FUNCTION_BLOCK "SEQUENCE"   // FB18, GRAPH_PLUS
{ S7_Optimized_Access := 'TRUE' }
VERSION : 0.1
   VAR_INPUT
      OFF_SQ : Bool := false;   // Turn sequence off
      INIT_SQ : Bool := false;   // Set sequence to initial state
      ACK_EF : Bool := false;   // Acknowledge all errors and faults
      S_PREV : Bool := false;   // Output previous step in parameter S_NO
      S_NEXT : Bool := false;   // Indicate next step in parameter S_NO
      SW_AUTO : Bool := false;   // Automatic mode
      SW_TAP : Bool := false;   // Semiautomatic/switch with transition
      SW_TOP : Bool := false;   // Semiautomatic/ignore transition
      SW_MAN : Bool := false;   // Manual mode
      S_SEL : Int := 0;   // Select step to be output to S_NO
      S_ON : Bool := false;   // Activate step indicated in S_NO
      S_OFF : Bool := false;   // Deactivate step indicated S_NO
      T_PUSH : Bool := false;   // Enable transition to switch in semi automatic mode
   END_VAR
   VAR_OUTPUT
      S_NO : Int := 0;   // Step number
      S_MORE : Bool := false;   // More steps are available and can be shown in S_NO
      S_ACTIVE : Bool := false;   // Step indicated in S_NO is active
      ERR_FLT : Bool := false;   // Interlock or supervision group error
      AUTO_ON : Bool := false;   // Automatic mode is active
      TAP_ON : Bool := false;   // Semiautomatic mode/step with transition enabled
      TOP_ON : Bool := false;   // Semiautomatic mode/ignore transition enabled
      MAN_ON : Bool := false;   // Manual mode is active
   END_VAR
   VAR
      HMI_INFO : Array[0..8] of UInt;
      IF_PAR : G7_IfParPlus_V2;
      RT_DATA : G7_RTDataPlus_V2;   // Internal data area
      Trans1 : G7_TransitionPlus_V2;   // Transition structure
      Trans2 : G7_TransitionPlus_V2;   // Transition structure
      Trans3 : G7_TransitionPlus_V2;   // Transition structure
      Trans4 : G7_TransitionPlus_V2;   // Transition structure
      Trans5 : G7_TransitionPlus_V2;   // Transition structure
      Idle : G7_StepPlus_V2;   // Step structure
      Warmup : G7_StepPlus_V2;   // Step structure
      Stabilize : G7_StepPlus_V2;   // Step structure
      Generation : G7_StepPlus_V2;   // Step structure
      Cooldown : G7_StepPlus_V2;   // Step structure
      SINI : Array[0..1] of USInt;
      LSTT : Array[0..4] of USInt;
      ATAJ : Array[0..4] of USInt;
      ATAB : Array[0..4] of USInt;
      PSTT : Array[0..4] of USInt;
      NSTT : Array[0..4] of USInt;
      ASSJ : Array[0..4] of USInt;
      ASSB : Array[0..4] of USInt;
      PTTS : Array[0..4] of USInt;
      NTTS : Array[0..4] of USInt;
      SW_SQTS : Array[0..4] of USInt;
      SWITCH : Array[0..0] of USInt;
      TVX : Array[0..1] of USInt;
      TTX : Array[0..1] of USInt;
      TSX : Array[0..1] of USInt;
      S00X : Array[0..1] of USInt;
      SOFFX : Array[0..1] of USInt;
      SONX : Array[0..1] of USInt;
      SAX : Array[0..1] of USInt;
      SERRX : Array[0..5] of USInt;
      SMX : Array[0..5] of USInt;
      S0X : Array[0..5] of USInt;
      S1X : Array[0..5] of USInt;
      IL_ALARM_INST : Program_Alarm;
      SUP_ALARM_INST : Program_Alarm;
      STEP_TIME_ALARM_INST : Program_Alarm;
      IEC_TIMER_INST : IEC_TIMER;
      TRANSACTION_FLAG : Bool := false;
   END_VAR
   // SINI[0] := 2;
   // LSTT[0] := 255;
   // LSTT[1] := 255;
   // LSTT[2] := 255;
   // LSTT[3] := 255;
   // ATAJ[1] := 1;
   // ATAJ[2] := 2;
   // ATAJ[3] := 3;
   // ATAJ[4] := 4;
   // ATAB[1] := 1;
   // ATAB[2] := 2;
   // ATAB[3] := 3;
   // ATAB[4] := 4;
   // PSTT[1] := 1;
   // PSTT[2] := 2;
   // PSTT[3] := 3;
   // PSTT[4] := 4;
   // NSTT[0] := 1;
   // NSTT[1] := 2;
   // NSTT[2] := 3;
   // NSTT[3] := 4;
   // ASSJ[1] := 1;
   // ASSJ[2] := 2;
   // ASSJ[3] := 3;
   // ASSJ[4] := 4;
   // ASSB[1] := 1;
   // ASSB[2] := 2;
   // ASSB[3] := 3;
   // ASSB[4] := 4;
   // PTTS[0] := 255;
   // PTTS[2] := 1;
   // PTTS[3] := 2;
   // PTTS[4] := 3;
   // NTTS[1] := 1;
   // NTTS[2] := 2;
   // NTTS[3] := 3;
   // NTTS[4] := 4;
   // TVX[0] := 16#1;
   // TTX[0] := 16#1;
   // TSX[0] := 16#1;
   // S00X[0] := 16#1;
   // SOFFX[0] := 16#1;
   // SONX[0] := 16#1;
   // SAX[0] := 16#1;
   // SERRX[0] := 16#1;
   // SMX[0] := 16#1;
   // S0X[0] := 16#1;
   // S1X[0] := 16#1;
BEGIN
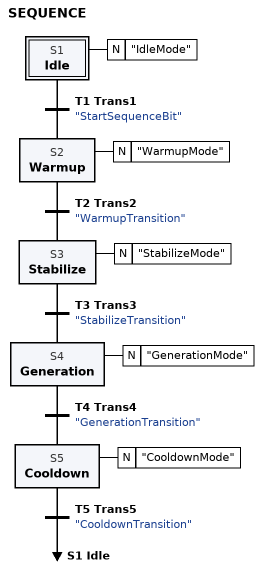
   // sequencer 1
   INITIAL_STEP Idle:   // S1, max time T#10S, warning time T#7S
              N    "IdleMode"
   END_STEP
   TRANSITION Trans1 FROM Idle TO Warmup   // T1
      := "StartSequenceBit";
   END_TRANSITION
   STEP Warmup:   // S2, max time T#10S, warning time T#7S
              N    "WarmupMode"
   END_STEP
   TRANSITION Trans2 FROM Warmup TO Stabilize   // T2
      := "WarmupTransition";
   END_TRANSITION
   STEP Stabilize:   // S3, max time T#10S, warning time T#7S
              N    "StabilizeMode"
   END_STEP
   TRANSITION Trans3 FROM Stabilize TO Generation   // T3
      := "StabilizeTransition";
   END_TRANSITION
   STEP Generation:   // S4, max time T#10S, warning time T#7S
              N    "GenerationMode"
   END_STEP
   TRANSITION Trans4 FROM Generation TO Cooldown   // T4
      := "GenerationTransition";
   END_TRANSITION
   STEP Cooldown:   // S5, max time T#10S, warning time T#7S
              N    "CooldownMode"
   END_STEP
   TRANSITION Trans5 FROM Cooldown TO Idle   // T5, jump
      := "CooldownTransition";
   END_TRANSITION
END_FUNCTION_BLOCK

FUNCTION_BLOCK "HOURMETER_LAD"   // FB19, LAD
{ S7_Optimized_Access := 'TRUE' }
VERSION : 0.1
   VAR
      Accum_Elapsed : Time;
      OS1 : Bool;
      MinuteTimedDown : Bool;
      HourCountedDown : Bool;
      OS2 : Bool;
      OS3 : Bool;
      DayCountedDown : Bool;
      ResetTime : Time;
      OS4 : Bool;
      ResetRTO : Bool;
      MinuteCounterReset : Bool;
      HourCounterReset : Bool;
   END_VAR
   VAR_TEMP
      ResetHourmeterTrigger : Bool;
   END_VAR
   VAR_TEMP   // added for the SCL form of the ladder/FBD networks
      _w1 : Bool;
      _w2 : Bool;
      _w3 : Bool;
   END_VAR
BEGIN

REGION Network 1
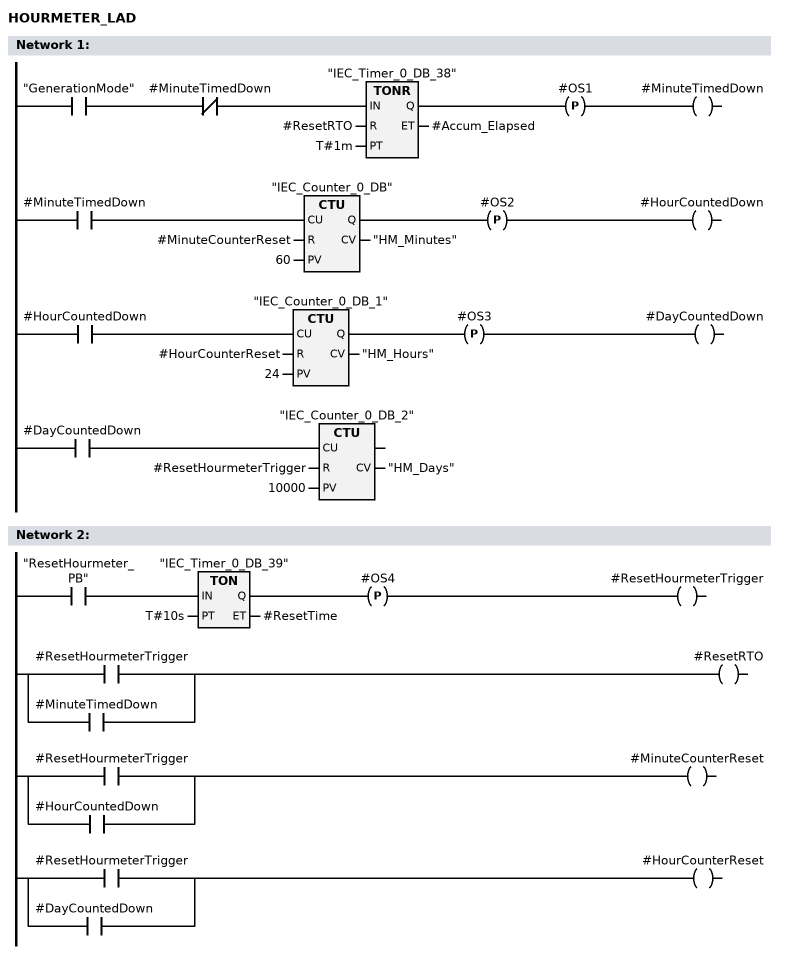
   "IEC_Timer_0_DB_38".TONR(IN := "GenerationMode" AND NOT #MinuteTimedDown,
                           R := #ResetRTO,
                           PT := T#1m,
                           ET => #Accum_Elapsed);
   #_w1 := "IEC_Timer_0_DB_38".Q AND NOT #OS1;   // rising edge
   #OS1 := "IEC_Timer_0_DB_38".Q;
   #MinuteTimedDown := #_w1;
   "IEC_Counter_0_DB".CTU(CU := #MinuteTimedDown, R := #MinuteCounterReset, PV := 60, CV => "HM_Minutes");
   #_w2 := "IEC_Counter_0_DB".Q AND NOT #OS2;   // rising edge
   #OS2 := "IEC_Counter_0_DB".Q;
   #HourCountedDown := #_w2;
   "IEC_Counter_0_DB_1".CTU(CU := #HourCountedDown, R := #HourCounterReset, PV := 24, CV => "HM_Hours");
   #_w3 := "IEC_Counter_0_DB_1".Q AND NOT #OS3;   // rising edge
   #OS3 := "IEC_Counter_0_DB_1".Q;
   #DayCountedDown := #_w3;
   "IEC_Counter_0_DB_2".CTU(CU := #DayCountedDown, R := #ResetHourmeterTrigger, PV := 10000, CV => "HM_Days");
END_REGION

REGION Network 2
   "IEC_Timer_0_DB_39".TON(IN := "ResetHourmeter_PB", PT := T#10s, ET => #ResetTime);
   #_w1 := "IEC_Timer_0_DB_39".Q AND NOT #OS4;   // rising edge
   #OS4 := "IEC_Timer_0_DB_39".Q;
   #ResetHourmeterTrigger := #_w1;
   #ResetRTO := #ResetHourmeterTrigger OR #MinuteTimedDown;
   #MinuteCounterReset := #ResetHourmeterTrigger OR #HourCountedDown;
   #HourCounterReset := #ResetHourmeterTrigger OR #DayCountedDown;
END_REGION
END_FUNCTION_BLOCK

FUNCTION_BLOCK "HOURMETER_FBD"   // FB20, FBD
{ S7_Optimized_Access := 'TRUE' }
VERSION : 0.1
   VAR
      Accum_Elapsed : Time;
      OS1 : Bool;
      MinuteTimedDown : Bool;
      HourCountedDown : Bool;
      OS2 : Bool;
      OS3 : Bool;
      DayCountedDown : Bool;
      ResetTime : Time;
      OS4 : Bool;
      ResetRTO : Bool;
      MinuteCounterReset : Bool;
      HourCounterReset : Bool;
   END_VAR
   VAR_TEMP
      ResetHourmeterTrigger : Bool;
   END_VAR
   VAR_TEMP   // added for the SCL form of the ladder/FBD networks
      _w1 : Bool;
      _w2 : Bool;
      _w3 : Bool;
   END_VAR
BEGIN

REGION Network 1
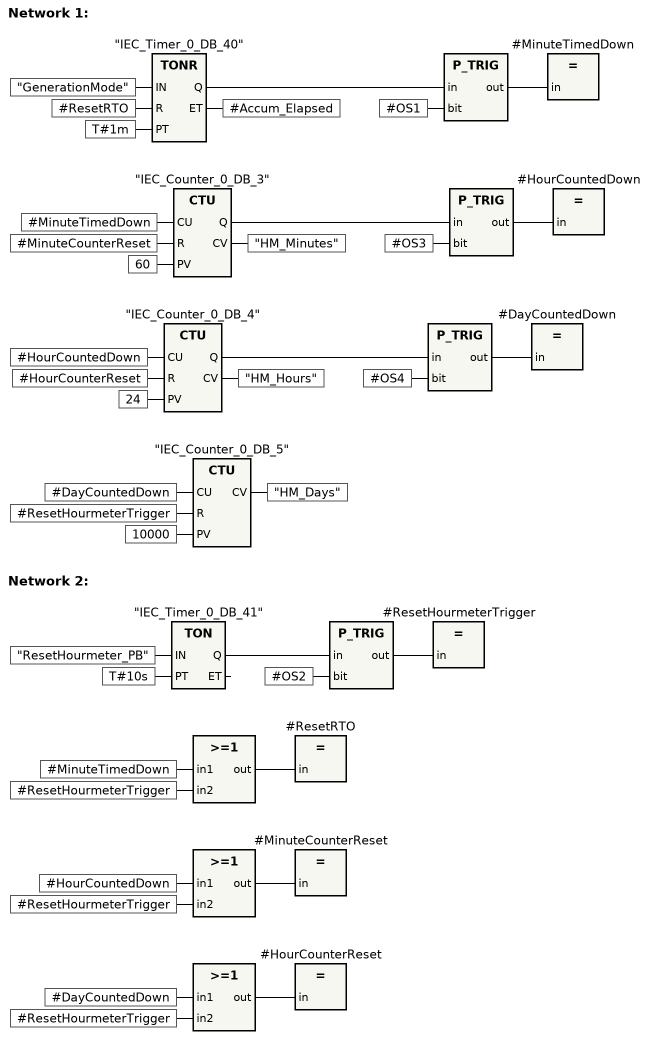
   "IEC_Timer_0_DB_40".TONR(IN := "GenerationMode", R := #ResetRTO, PT := T#1m, ET => #Accum_Elapsed);
   #_w1 := "IEC_Timer_0_DB_40".Q AND NOT #OS1;   // rising edge
   #OS1 := "IEC_Timer_0_DB_40".Q;
   #MinuteTimedDown := #_w1;
   "IEC_Counter_0_DB_3".CTU(CU := #MinuteTimedDown, R := #MinuteCounterReset, PV := 60, CV => "HM_Minutes");
   #_w2 := "IEC_Counter_0_DB_3".Q AND NOT #OS3;   // rising edge
   #OS3 := "IEC_Counter_0_DB_3".Q;
   #HourCountedDown := #_w2;
   "IEC_Counter_0_DB_4".CTU(CU := #HourCountedDown, R := #HourCounterReset, PV := 24, CV => "HM_Hours");
   #_w3 := "IEC_Counter_0_DB_4".Q AND NOT #OS4;   // rising edge
   #OS4 := "IEC_Counter_0_DB_4".Q;
   #DayCountedDown := #_w3;
   "IEC_Counter_0_DB_5".CTU(CU := #DayCountedDown, R := #ResetHourmeterTrigger, PV := 10000, CV => "HM_Days");
END_REGION

REGION Network 2
   "IEC_Timer_0_DB_41".TON(IN := "ResetHourmeter_PB", PT := T#10s);
   #_w1 := "IEC_Timer_0_DB_41".Q AND NOT #OS2;   // rising edge
   #OS2 := "IEC_Timer_0_DB_41".Q;
   #ResetHourmeterTrigger := #_w1;
   #ResetRTO := #MinuteTimedDown OR #ResetHourmeterTrigger;
   #MinuteCounterReset := #HourCountedDown OR #ResetHourmeterTrigger;
   #HourCounterReset := #DayCountedDown OR #ResetHourmeterTrigger;
END_REGION
END_FUNCTION_BLOCK

FUNCTION_BLOCK "HOURMETER_SCL"   // FB21, SCL
{ S7_Optimized_Access := 'TRUE' }
VERSION : 0.1
   VAR
      Accum_Elapsed : Time;
      OS1 : Bool;
      MinuteTimedDown : Bool;
      HourCountedDown : Bool;
      OS2 : Bool;
      OS3 : Bool;
      DayCountedDown : Bool;
      ResetTime : Time;
      OS4 : Bool;
      ResetRTO : Bool;
      MinuteCounterReset : Bool;
      HourCounterReset : Bool;
   END_VAR
   VAR_TEMP
      ResetHourmeterTrigger : Bool;
   END_VAR
BEGIN
   IF "GenerationMode" THEN
       "IEC_Timer_0_DB_43".TONR(IN := TRUE,
                                R := #ResetRTO,
                                PT := T#60s,
                                Q => #MinuteTimedDown,
                                ET => #Accum_Elapsed);
   END_IF;

   IF #MinuteTimedDown THEN
       RESET_TIMER("IEC_Timer_0_DB_43");
   END_IF;

   "IEC_Counter_0_DB_6".CTU(CU:=#MinuteTimedDown,
                            R:=#MinuteCounterReset,
                            PV:=60,
                            Q=>#HourCountedDown,
                            CV=>"HM_Minutes");

   "IEC_Counter_0_DB_7".CTU(CU:=#HourCountedDown,
                            R:=#HourCounterReset,
                            PV:=24,
                            Q=>#DayCountedDown,
                            CV=>"HM_Hours");

   "IEC_Counter_0_DB_8".CTU(CU:=#DayCountedDown,
                            R:=#ResetHourmeterTrigger,
                            PV:=10000,
                            CV=>"HM_Days");

   IF "ResetHourmeter_PB" THEN
       "IEC_Timer_0_DB_44".TON(IN := TRUE,
                               PT := T#10s,
                               Q => #ResetHourmeterTrigger);
   ELSE
       RESET_TIMER("IEC_Timer_0_DB_44");
   END_IF;

   IF #ResetHourmeterTrigger OR #MinuteTimedDown THEN
       #ResetRTO := 1;
   ELSE
       #ResetRTO := 0;
   END_IF;

   IF #ResetHourmeterTrigger OR #HourCountedDown THEN
       #MinuteCounterReset := 1;
   ELSE
       #MinuteCounterReset := 0;
   END_IF;

   IF #ResetHourmeterTrigger OR #DayCountedDown THEN
       #HourCounterReset := 1;
   ELSE
       #HourCounterReset := 0;
   END_IF;
END_FUNCTION_BLOCK

FUNCTION_BLOCK "HOURMETER_STL"   // FB22, STL
{ S7_Optimized_Access := 'TRUE' }
VERSION : 0.1
   VAR
      Accum_Elapsed : Time;
      OS1 : Bool;
      MinuteTimedDown : Bool;
      HourCountedDown : Bool;
      OS2 : Bool;
      OS3 : Bool;
      DayCountedDown : Bool;
      ResetTime : Time;
      OS4 : Bool;
      ResetRTO : Bool;
      MinuteCounterReset : Bool;
      HourCounterReset : Bool;
   END_VAR
   VAR_TEMP
      ResetHourmeterTrigger : Bool;
      TooManyDays : Bool;
      Acc_Time : Time;
   END_VAR
BEGIN

REGION Network 1
         A     "GenerationMode";
         JC    RTOTimer;
         CLR;
         JU    EndOfLine;

   RTOTimer:CALL  TONR, "IEC_Timer_0_DB_45"
         ( IN := TRUE,
           R  := #ResetRTO,
           PT := T#1m,
           Q  := #MinuteTimedDown,
           ET := #Accum_Elapsed
         );

         CALL  CTU, "IEC_Counter_0_DB_9"
         ( CU := #MinuteTimedDown,
           R  := #MinuteCounterReset,
           PV := 60,
           Q  := #HourCountedDown,
           CV := "HM_Minutes"
         );

         CALL  CTU, "IEC_Counter_0_DB_10"
         ( CU := #HourCountedDown,
           R  := #HourCounterReset,
           PV := 24,
           Q  := #DayCountedDown,
           CV := "HM_Hours"
         );

         CALL  CTU, "IEC_Counter_0_DB_11"
         ( CU := #DayCountedDown,
           R  := #ResetHourmeterTrigger,
           PV := 10000,
           Q  := #TooManyDays,
           CV := "HM_Days"
         );

         JU    EndOfLine;



   ResetEvaluate:CLR;
         A     "ResetHourmeter_PB";
         JC    ResetHourmeter;
         CALL  RESET_TIMER
         ( "TIMER" := "IEC_Timer_0_DB_46"
         );
         JU    EndOfLine;

   ResetHourmeter:CALL  TON, "IEC_Timer_0_DB_46"
         ( IN := TRUE,
           PT := T#10s,
           Q  := #ResetHourmeterTrigger,
           ET := #Acc_Time
         );

   EndOfLine:A     #ResetHourmeterTrigger;
         O     #MinuteTimedDown;
         =     #ResetRTO;
         CLR;
         A     #ResetHourmeterTrigger;
         O     #HourCountedDown;
         =     #MinuteCounterReset;
         CLR;
         A     #ResetHourmeterTrigger;
         O     #DayCountedDown;
         =     #HourCountedDown;
END_REGION
END_FUNCTION_BLOCK

FUNCTION "SCP" : Void   // FC1, FBD
{ S7_Optimized_Access := 'TRUE' }
VERSION : 0.1
   VAR_INPUT
      Input_Min : Int;
      Input_Max : Int;
      Input_Signal : Int;
      Output_Min : Int;
      Output_Max : Int;
   END_VAR
   VAR_OUTPUT
      SV : Int;
   END_VAR
   VAR_TEMP
      TV : Real;
   END_VAR
BEGIN

REGION Network 1
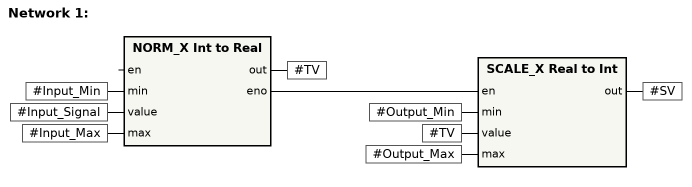
   #TV := NORM_X(MIN := #Input_Min, VALUE := #Input_Signal, MAX := #Input_Max);
   #SV := SCALE_X(MIN := #Output_Min, VALUE := #TV, MAX := #Output_Max);
END_REGION
END_FUNCTION

FUNCTION "MOVE" : Void   // FC2, FBD
{ S7_Optimized_Access := 'TRUE' }
VERSION : 0.1
   VAR_INPUT
      Int1 : Int;
   END_VAR
   VAR_OUTPUT
      Time1 : Time;
   END_VAR
   VAR_TEMP
      TV : Int;
   END_VAR
BEGIN

REGION Network 1
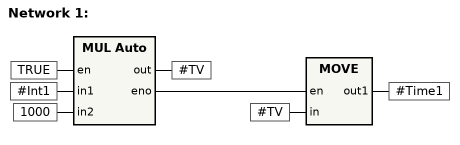
   IF TRUE THEN
       #TV := #Int1 * 1000;
       #Time1 := #TV;
   END_IF;
END_REGION
END_FUNCTION

ORGANIZATION_BLOCK "Main"   // OB1, LAD, ProgramCycle
TITLE = "Main Program Sweep (Cycle)"
{ S7_Optimized_Access := 'TRUE' }
VERSION : 0.1
   VAR_INPUT
      Initial_Call : Bool;   // Initial call of this OB
      Remanence : Bool;   // =True, if remanent data are available
   END_VAR
   VAR_TEMP
      SequenceInit : Bool;
      InitSequence : Bool;
   END_VAR
   VAR_TEMP   // added for the SCL form of the ladder/FBD networks
      _w1 : Bool;
      _w2 : Bool;
      _w3 : Bool;
      _w4 : Bool;
   END_VAR
BEGIN

REGION Network 1
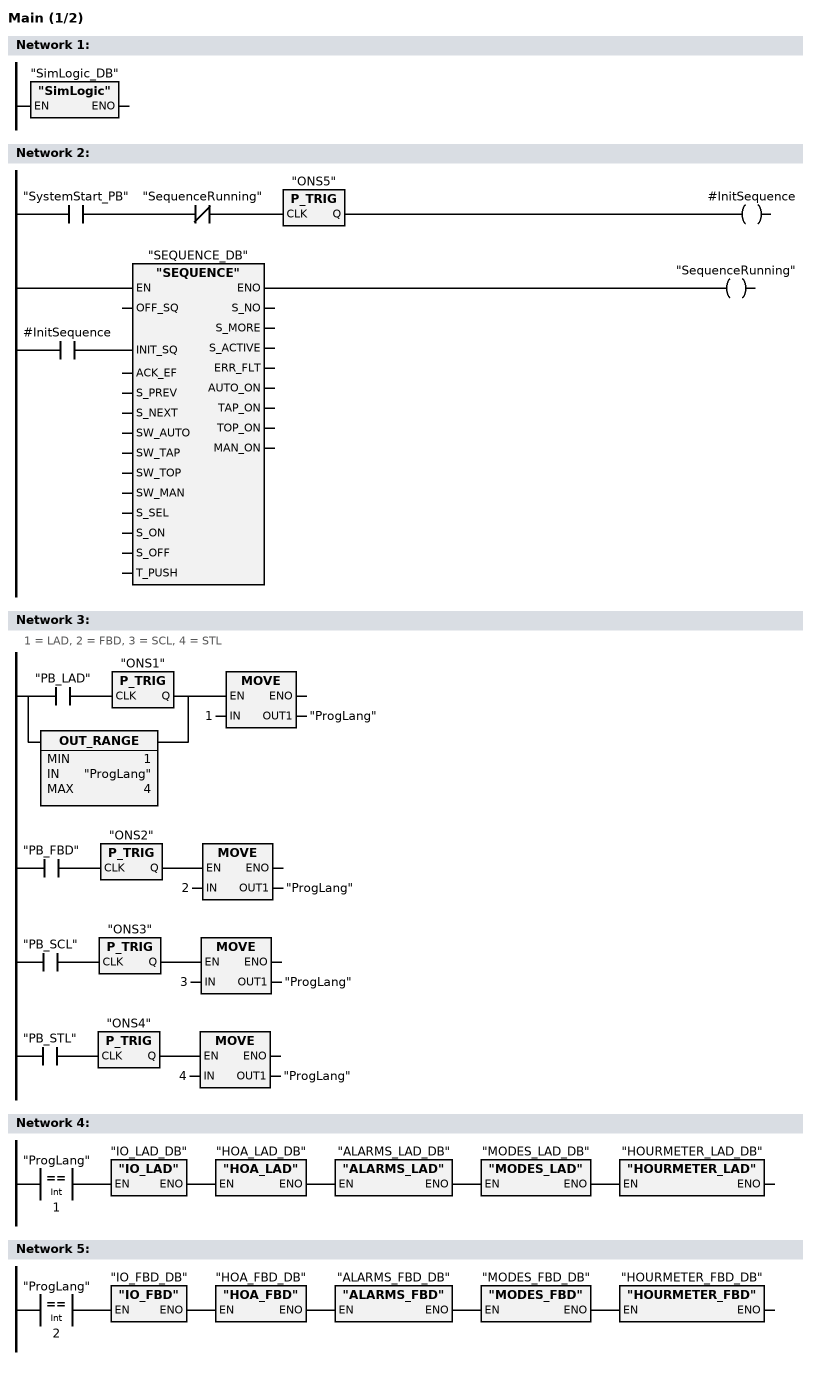
   RUNG wire#powerrail
      "SimLogic_DB"()
   END_RUNG
   // the same network as SCL:
   "SimLogic_DB"();   // "SimLogic"
END_REGION

REGION Network 2
   RUNG wire#powerrail
      Contact( "SystemStart_PB" )
      I_Contact( "SequenceRunning" )
      P_Trig( "ONS5" )
      Coil( #InitSequence )
   END_RUNG
   RUNG wire#powerrail
      "SEQUENCE_DB"(INIT_SQ := wire#w1, OFF_SQ :=, ACK_EF :=, S_PREV :=, S_NEXT :=, SW_AUTO :=, SW_TAP :=, SW_TOP :=, SW_MAN :=, S_SEL :=, S_ON :=, S_OFF :=, T_PUSH :=, S_NO =>, S_MORE =>, S_ACTIVE =>, ERR_FLT =>, AUTO_ON =>, TAP_ON =>, TOP_ON =>, MAN_ON =>)
      Coil( "SequenceRunning" )
   END_RUNG
   RUNG wire#powerrail
      Contact( #InitSequence )
   END_RUNG wire#w1
   // the same network as SCL:
   #_w1 := "SystemStart_PB" AND NOT "SequenceRunning";
   #_w2 := #_w1 AND NOT "ONS5";   // rising edge
   "ONS5" := #_w1;
   #InitSequence := #_w2;
   "SEQUENCE_DB"(INIT_SQ := #InitSequence, ENO => #_w3);   // "SEQUENCE"
   "SequenceRunning" := #_w3;
END_REGION

REGION Network 3
   // 1 = LAD, 2 = FBD, 3 = SCL, 4 = STL
   #_w1 := "PB_LAD" AND NOT "ONS1";   // rising edge
   "ONS1" := "PB_LAD";
   IF #_w1 OR ("ProgLang" < 1) OR ("ProgLang" > 4) THEN "ProgLang" := 1; END_IF;
   #_w2 := "PB_FBD" AND NOT "ONS2";   // rising edge
   "ONS2" := "PB_FBD";
   IF #_w2 THEN "ProgLang" := 2; END_IF;
   #_w3 := "PB_SCL" AND NOT "ONS3";   // rising edge
   "ONS3" := "PB_SCL";
   IF #_w3 THEN "ProgLang" := 3; END_IF;
   #_w4 := "PB_STL" AND NOT "ONS4";   // rising edge
   "ONS4" := "PB_STL";
   IF #_w4 THEN "ProgLang" := 4; END_IF;
END_REGION

REGION Network 4
   RUNG wire#powerrail
      { S7_Templates := "SrcType := Int" } EQ_Contact(in1 := "ProgLang", in2 := 1)
      "IO_LAD_DB"()
      "HOA_LAD_DB"()
      "ALARMS_LAD_DB"()
      "MODES_LAD_DB"()
      "HOURMETER_LAD_DB"()
   END_RUNG
   // the same network as SCL:
   "IO_LAD_DB"(EN := "ProgLang" = 1, ENO => #_w1);   // "IO_LAD"
   "HOA_LAD_DB"(EN := #_w1, ENO => #_w2);   // "HOA_LAD"
   "ALARMS_LAD_DB"(EN := #_w2, ENO => #_w3);   // "ALARMS_LAD"
   "MODES_LAD_DB"(EN := #_w3, ENO => #_w4);   // "MODES_LAD"
   IF #_w4 THEN
       "HOURMETER_LAD_DB"();   // "HOURMETER_LAD"
   END_IF;
END_REGION

REGION Network 5
   RUNG wire#powerrail
      { S7_Templates := "SrcType := Int" } EQ_Contact(in1 := "ProgLang", in2 := 2)
      "IO_FBD_DB"()
      "HOA_FBD_DB"()
      "ALARMS_FBD_DB"()
      "MODES_FBD_DB"()
      "HOURMETER_FBD_DB"()
   END_RUNG
   // the same network as SCL:
   "IO_FBD_DB"(EN := "ProgLang" = 2, ENO => #_w1);   // "IO_FBD"
   "HOA_FBD_DB"(EN := #_w1, ENO => #_w2);   // "HOA_FBD"
   "ALARMS_FBD_DB"(EN := #_w2, ENO => #_w3);   // "ALARMS_FBD"
   "MODES_FBD_DB"(EN := #_w3, ENO => #_w4);   // "MODES_FBD"
   IF #_w4 THEN
       "HOURMETER_FBD_DB"();   // "HOURMETER_FBD"
   END_IF;
END_REGION

REGION Network 6
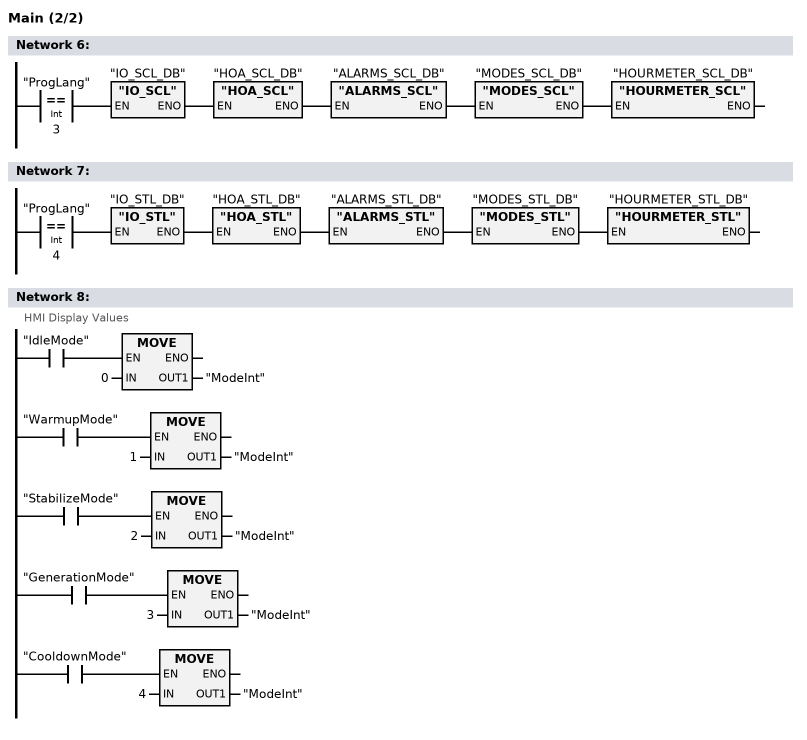
   RUNG wire#powerrail
      { S7_Templates := "SrcType := Int" } EQ_Contact(in1 := "ProgLang", in2 := 3)
      "IO_SCL_DB"()
      "HOA_SCL_DB"()
      "ALARMS_SCL_DB"()
      "MODES_SCL_DB"()
      "HOURMETER_SCL_DB"()
   END_RUNG
   // the same network as SCL:
   "IO_SCL_DB"(EN := "ProgLang" = 3, ENO => #_w1);   // "IO_SCL"
   "HOA_SCL_DB"(EN := #_w1, ENO => #_w2);   // "HOA_SCL"
   "ALARMS_SCL_DB"(EN := #_w2, ENO => #_w3);   // "ALARMS_SCL"
   "MODES_SCL_DB"(EN := #_w3, ENO => #_w4);   // "MODES_SCL"
   IF #_w4 THEN
       "HOURMETER_SCL_DB"();   // "HOURMETER_SCL"
   END_IF;
END_REGION

REGION Network 7
   RUNG wire#powerrail
      { S7_Templates := "SrcType := Int" } EQ_Contact(in1 := "ProgLang", in2 := 4)
      "IO_STL_DB"()
      "HOA_STL_DB"()
      "ALARMS_STL_DB"()
      "MODES_STL_DB"()
      "HOURMETER_STL_DB"()
   END_RUNG
   // the same network as SCL:
   "IO_STL_DB"(EN := "ProgLang" = 4, ENO => #_w1);   // "IO_STL"
   "HOA_STL_DB"(EN := #_w1, ENO => #_w2);   // "HOA_STL"
   "ALARMS_STL_DB"(EN := #_w2, ENO => #_w3);   // "ALARMS_STL"
   "MODES_STL_DB"(EN := #_w3, ENO => #_w4);   // "MODES_STL"
   IF #_w4 THEN
       "HOURMETER_STL_DB"();   // "HOURMETER_STL"
   END_IF;
END_REGION

REGION Network 8
   // HMI Display Values
   RUNG wire#powerrail
      Contact( "IdleMode" )
      Move(in := 0, out1 => "ModeInt")
   END_RUNG
   RUNG wire#powerrail
      Contact( "WarmupMode" )
      Move(in := 1, out1 => "ModeInt")
   END_RUNG
   RUNG wire#powerrail
      Contact( "StabilizeMode" )
      Move(in := 2, out1 => "ModeInt")
   END_RUNG
   RUNG wire#powerrail
      Contact( "GenerationMode" )
      Move(in := 3, out1 => "ModeInt")
   END_RUNG
   RUNG wire#powerrail
      Contact( "CooldownMode" )
      Move(in := 4, out1 => "ModeInt")
   END_RUNG
   // the same network as SCL:
   IF "IdleMode" THEN "ModeInt" := 0; END_IF;
   IF "WarmupMode" THEN "ModeInt" := 1; END_IF;
   IF "StabilizeMode" THEN "ModeInt" := 2; END_IF;
   IF "GenerationMode" THEN "ModeInt" := 3; END_IF;
   IF "CooldownMode" THEN "ModeInt" := 4; END_IF;
END_REGION
END_ORGANIZATION_BLOCK

ORGANIZATION_BLOCK "PID"   // OB30, LAD, CyclicInterrupt
{ S7_Optimized_Access := 'TRUE' }
VERSION : 0.1
   VAR_INPUT
      Initial_Call : Bool;   // Initial call of this OB
      Event_Count : Int;   // Events discarded
   END_VAR
   VAR_TEMP
      BSP : Real;
      VSP : Real;
      BaffleHandTrigger : Bool;
      BaffleAutoTrigger : Bool;
      BaffleOffTrigger : Bool;
      VFDHandTrigger : Bool;
      VFDOffTrigger : Bool;
      VFDAutoTrigger : Bool;
   END_VAR
   VAR_TEMP   // added for the SCL form of the ladder/FBD networks
      _w1 : Bool;
      _w2 : Bool;
      _w3 : Bool;
      _w4 : Bool;
      _w5 : Bool;
      _w6 : Bool;
      _w7 : Bool;
   END_VAR
BEGIN

REGION Network 1: Oil High Flow Alarm Handling
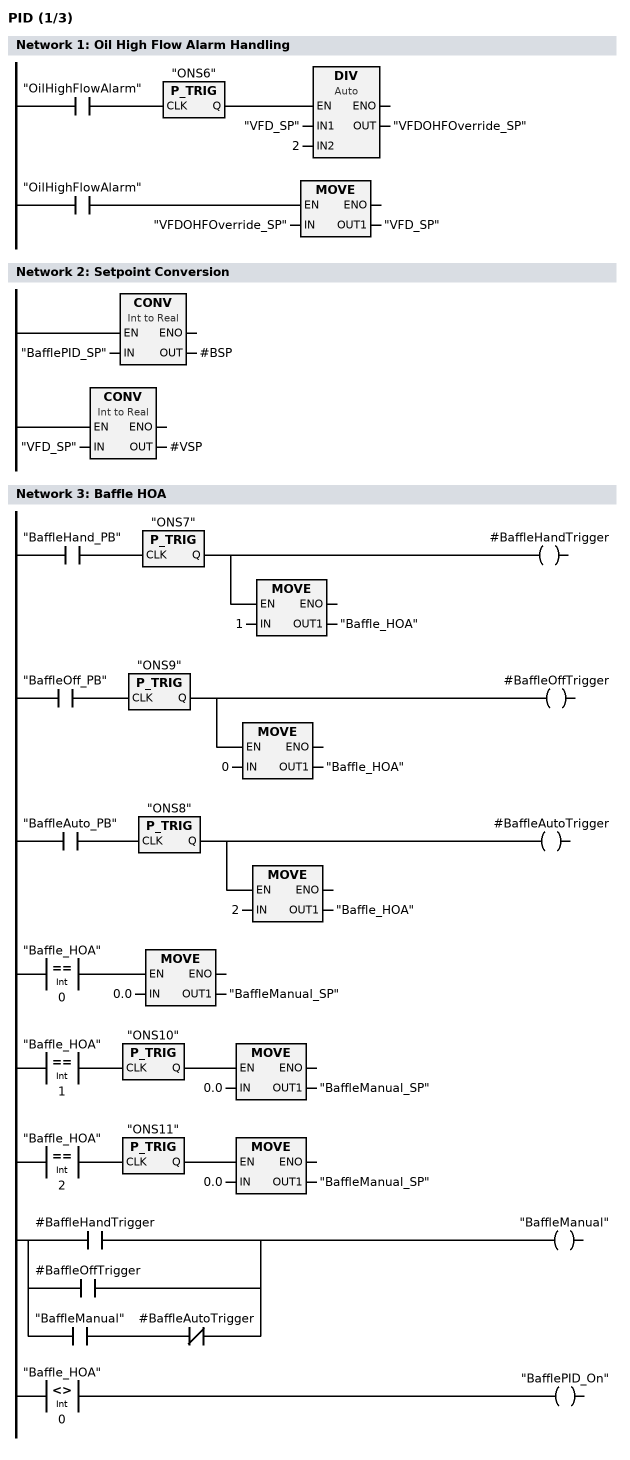
   RUNG wire#powerrail
      Contact( "OilHighFlowAlarm" )
      P_Trig( "ONS6" )
      Div(in1 := "VFD_SP", in2 := 2, out => "VFDOHFOverride_SP")
   END_RUNG
   RUNG wire#powerrail
      Contact( "OilHighFlowAlarm" )
      Move(in := "VFDOHFOverride_SP", out1 => "VFD_SP")
   END_RUNG
   // the same network as SCL:
   #_w1 := "OilHighFlowAlarm" AND NOT "ONS6";   // rising edge
   "ONS6" := "OilHighFlowAlarm";
   IF #_w1 THEN "VFDOHFOverride_SP" := "VFD_SP" / 2; END_IF;
   IF "OilHighFlowAlarm" THEN "VFD_SP" := "VFDOHFOverride_SP"; END_IF;
END_REGION

REGION Network 2: Setpoint Conversion
   RUNG wire#powerrail
      { S7_Templates := "[SrcType := Int, DestType := Real]" } Convert(in := "BafflePID_SP", out => #BSP)
   END_RUNG
   RUNG wire#powerrail
      { S7_Templates := "[SrcType := Int, DestType := Real]" } Convert(in := "VFD_SP", out => #VSP)
   END_RUNG
   // the same network as SCL:
   #BSP := INT_TO_REAL("BafflePID_SP");
   #VSP := INT_TO_REAL("VFD_SP");
END_REGION

REGION Network 3: Baffle HOA
   RUNG wire#powerrail
      Contact( "BaffleHand_PB" )
      P_Trig( "ONS7" )
      wire#w1
      Coil( #BaffleHandTrigger )
   END_RUNG
   RUNG wire#w1
      Move(in := 1, out1 => "Baffle_HOA")
   END_RUNG
   RUNG wire#powerrail
      Contact( "BaffleOff_PB" )
      P_Trig( "ONS9" )
      wire#w2
      Coil( #BaffleOffTrigger )
   END_RUNG
   RUNG wire#w2
      Move(in := 0, out1 => "Baffle_HOA")
   END_RUNG
   RUNG wire#powerrail
      Contact( "BaffleAuto_PB" )
      P_Trig( "ONS8" )
      wire#w3
      Coil( #BaffleAutoTrigger )
   END_RUNG
   RUNG wire#w3
      Move(in := 2, out1 => "Baffle_HOA")
   END_RUNG
   RUNG wire#powerrail
      { S7_Templates := "SrcType := Int" } EQ_Contact(in1 := "Baffle_HOA", in2 := 0)
      Move(in := 0.0, out1 => "BaffleManual_SP")
   END_RUNG
   RUNG wire#powerrail
      { S7_Templates := "SrcType := Int" } EQ_Contact(in1 := "Baffle_HOA", in2 := 1)
      P_Trig( "ONS10" )
      Move(in := 0.0, out1 => "BaffleManual_SP")
   END_RUNG
   RUNG wire#powerrail
      { S7_Templates := "SrcType := Int" } EQ_Contact(in1 := "Baffle_HOA", in2 := 2)
      P_Trig( "ONS11" )
      Move(in := 0.0, out1 => "BaffleManual_SP")
   END_RUNG
   RUNG wire#powerrail
      Contact( #BaffleHandTrigger )
      wire#w4
      Coil( "BaffleManual" )
   END_RUNG
   RUNG wire#powerrail
      Contact( #BaffleOffTrigger )
   END_RUNG wire#w4
   RUNG wire#powerrail
      Contact( "BaffleManual" )
      I_Contact( #BaffleAutoTrigger )
   END_RUNG wire#w4
   RUNG wire#powerrail
      { S7_Templates := "SrcType := Int" } NE_Contact(in1 := "Baffle_HOA", in2 := 0)
      Coil( "BafflePID_On" )
   END_RUNG
   // the same network as SCL:
   #_w1 := "BaffleHand_PB" AND NOT "ONS7";   // rising edge
   "ONS7" := "BaffleHand_PB";
   #BaffleHandTrigger := #_w1;
   IF #_w1 THEN "Baffle_HOA" := 1; END_IF;
   #_w2 := "BaffleOff_PB" AND NOT "ONS9";   // rising edge
   "ONS9" := "BaffleOff_PB";
   #BaffleOffTrigger := #_w2;
   IF #_w2 THEN "Baffle_HOA" := 0; END_IF;
   #_w3 := "BaffleAuto_PB" AND NOT "ONS8";   // rising edge
   "ONS8" := "BaffleAuto_PB";
   #BaffleAutoTrigger := #_w3;
   IF #_w3 THEN "Baffle_HOA" := 2; END_IF;
   IF "Baffle_HOA" = 0 THEN "BaffleManual_SP" := 0.0; END_IF;
   #_w4 := "Baffle_HOA" = 1;
   #_w5 := #_w4 AND NOT "ONS10";   // rising edge
   "ONS10" := #_w4;
   IF #_w5 THEN "BaffleManual_SP" := 0.0; END_IF;
   #_w6 := "Baffle_HOA" = 2;
   #_w7 := #_w6 AND NOT "ONS11";   // rising edge
   "ONS11" := #_w6;
   IF #_w7 THEN "BaffleManual_SP" := 0.0; END_IF;
   "BaffleManual" := #BaffleHandTrigger OR #BaffleOffTrigger OR ("BaffleManual" AND NOT #BaffleAutoTrigger);
   "BafflePID_On" := "Baffle_HOA" <> 0;
END_REGION

REGION Network 4: VFD HOA
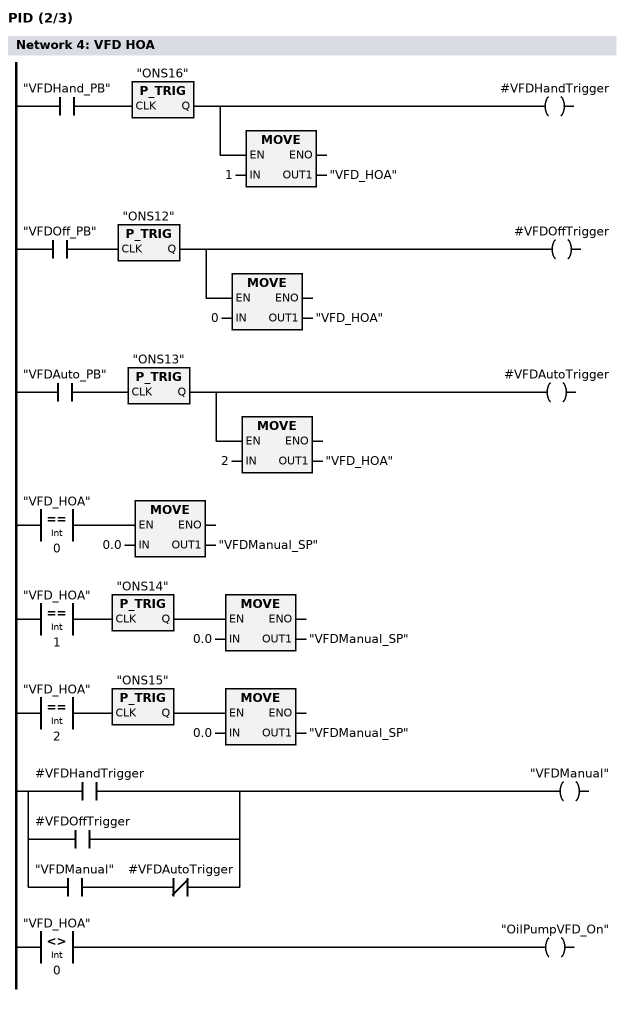
   RUNG wire#powerrail
      Contact( "VFDHand_PB" )
      P_Trig( "ONS16" )
      wire#w1
      Coil( #VFDHandTrigger )
   END_RUNG
   RUNG wire#w1
      Move(in := 1, out1 => "VFD_HOA")
   END_RUNG
   RUNG wire#powerrail
      Contact( "VFDOff_PB" )
      P_Trig( "ONS12" )
      wire#w2
      Coil( #VFDOffTrigger )
   END_RUNG
   RUNG wire#w2
      Move(in := 0, out1 => "VFD_HOA")
   END_RUNG
   RUNG wire#powerrail
      Contact( "VFDAuto_PB" )
      P_Trig( "ONS13" )
      wire#w3
      Coil( #VFDAutoTrigger )
   END_RUNG
   RUNG wire#w3
      Move(in := 2, out1 => "VFD_HOA")
   END_RUNG
   RUNG wire#powerrail
      { S7_Templates := "SrcType := Int" } EQ_Contact(in1 := "VFD_HOA", in2 := 0)
      Move(in := 0.0, out1 => "VFDManual_SP")
   END_RUNG
   RUNG wire#powerrail
      { S7_Templates := "SrcType := Int" } EQ_Contact(in1 := "VFD_HOA", in2 := 1)
      P_Trig( "ONS14" )
      Move(in := 0.0, out1 => "VFDManual_SP")
   END_RUNG
   RUNG wire#powerrail
      { S7_Templates := "SrcType := Int" } EQ_Contact(in1 := "VFD_HOA", in2 := 2)
      P_Trig( "ONS15" )
      Move(in := 0.0, out1 => "VFDManual_SP")
   END_RUNG
   RUNG wire#powerrail
      Contact( #VFDHandTrigger )
      wire#w4
      Coil( "VFDManual" )
   END_RUNG
   RUNG wire#powerrail
      Contact( #VFDOffTrigger )
   END_RUNG wire#w4
   RUNG wire#powerrail
      Contact( "VFDManual" )
      I_Contact( #VFDAutoTrigger )
   END_RUNG wire#w4
   RUNG wire#powerrail
      { S7_Templates := "SrcType := Int" } NE_Contact(in1 := "VFD_HOA", in2 := 0)
      Coil( "OilPumpVFD_On" )
   END_RUNG
   // the same network as SCL:
   #_w1 := "VFDHand_PB" AND NOT "ONS16";   // rising edge
   "ONS16" := "VFDHand_PB";
   #VFDHandTrigger := #_w1;
   IF #_w1 THEN "VFD_HOA" := 1; END_IF;
   #_w2 := "VFDOff_PB" AND NOT "ONS12";   // rising edge
   "ONS12" := "VFDOff_PB";
   #VFDOffTrigger := #_w2;
   IF #_w2 THEN "VFD_HOA" := 0; END_IF;
   #_w3 := "VFDAuto_PB" AND NOT "ONS13";   // rising edge
   "ONS13" := "VFDAuto_PB";
   #VFDAutoTrigger := #_w3;
   IF #_w3 THEN "VFD_HOA" := 2; END_IF;
   IF "VFD_HOA" = 0 THEN "VFDManual_SP" := 0.0; END_IF;
   #_w4 := "VFD_HOA" = 1;
   #_w5 := #_w4 AND NOT "ONS14";   // rising edge
   "ONS14" := #_w4;
   IF #_w5 THEN "VFDManual_SP" := 0.0; END_IF;
   #_w6 := "VFD_HOA" = 2;
   #_w7 := #_w6 AND NOT "ONS15";   // rising edge
   "ONS15" := #_w6;
   IF #_w7 THEN "VFDManual_SP" := 0.0; END_IF;
   "VFDManual" := #VFDHandTrigger OR #VFDOffTrigger OR ("VFDManual" AND NOT #VFDAutoTrigger);
   "OilPumpVFD_On" := "VFD_HOA" <> 0;
END_REGION

REGION Network 5
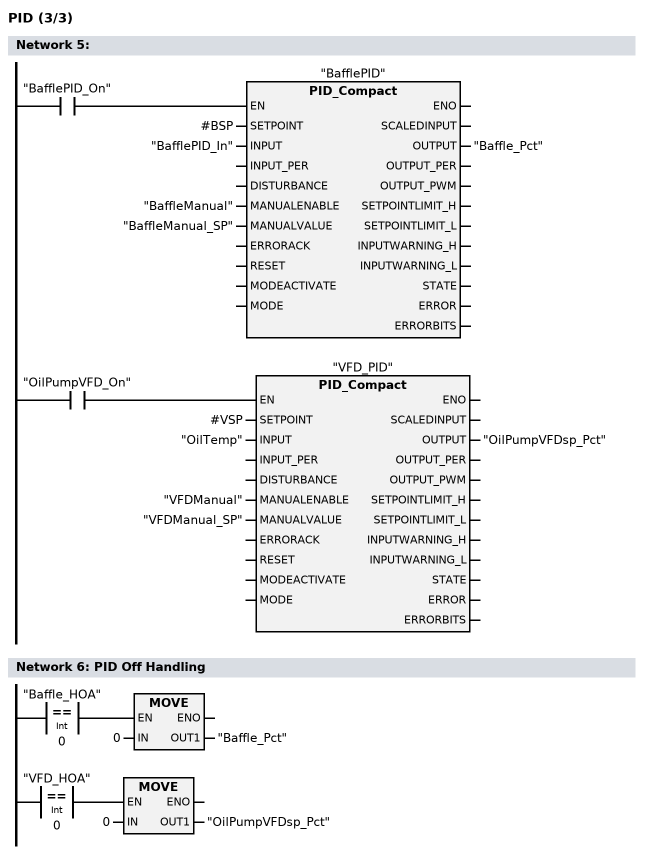
   IF "BafflePID_On" THEN
       "BafflePID"(Setpoint := #BSP,   // PID_Compact
                   Input := "BafflePID_In",
                   ManualEnable := "BaffleManual",
                   ManualValue := "BaffleManual_SP",
                   Output => "Baffle_Pct");
   END_IF;
   IF "OilPumpVFD_On" THEN
       "VFD_PID"(Setpoint := #VSP,   // PID_Compact
                 Input := "OilTemp",
                 ManualEnable := "VFDManual",
                 ManualValue := "VFDManual_SP",
                 Output => "OilPumpVFDsp_Pct");
   END_IF;
END_REGION

REGION Network 6: PID Off Handling
   RUNG wire#powerrail
      { S7_Templates := "SrcType := Int" } EQ_Contact(in1 := "Baffle_HOA", in2 := 0)
      Move(in := 0, out1 => "Baffle_Pct")
   END_RUNG
   RUNG wire#powerrail
      { S7_Templates := "SrcType := Int" } EQ_Contact(in1 := "VFD_HOA", in2 := 0)
      Move(in := 0, out1 => "OilPumpVFDsp_Pct")
   END_RUNG
   // the same network as SCL:
   IF "Baffle_HOA" = 0 THEN "Baffle_Pct" := 0; END_IF;
   IF "VFD_HOA" = 0 THEN "OilPumpVFDsp_Pct" := 0; END_IF;
END_REGION
END_ORGANIZATION_BLOCK

(* ===== HMI "HMI_RT_1" =====
system functions are stored by id; their names below are inferred from use
connection "1500PLC": S71200_TCP_IP, SCADA_S7_1500_OMS

HMI tags "Default tag table"
   "SystemStart_PB" : Bool = PLC SystemStart_PB AT %M63.1, 500 ms
   "SystemStop_PB" : Bool = PLC SystemStop_PB AT %M63.3, 500 ms
   "EStopAlarm" : Bool = PLC EStopAlarm AT %M41.6, 500 ms
   "BrakeFailureAlarm" : Bool = PLC BrakeFailureAlarm AT %M41.3, 500 ms
   "RotorOverspeedAlarm" : Bool = PLC RotorOverspeedAlarm AT %M40.7, 500 ms
   "OvercurrentAlarm" : Bool = PLC OvercurrentAlarm AT %M40.3, 500 ms
   "HighOilTempAlarm" : Bool = PLC HighOilTempAlarm AT %M40.5, 500 ms
   "OilLowFlowAlarm" : Bool = PLC OilLowFlowAlarm AT %M40.1, 500 ms
   "OilHighFlowAlarm" : Bool = PLC OilHighFlowAlarm AT %M41.1, 500 ms
   "AlarmSilence_PB" : Bool = PLC AlarmSilence_PB AT %M62.1, 500 ms
   "AlarmReset_PB" : Bool = PLC AlarmReset_PB AT %M62.0, 500 ms
   "Brake_En" : Bool = PLC Brake_Out AT %M0.0, 500 ms
   "StationInt_En" : Bool = PLC StationInterlock_Out AT %M1.5, 500 ms
   "VFD_En" : Bool = PLC OilPumpVFDen_Out AT %M0.2, 500 ms
   "Baffle_En" : Bool = PLC Baffle_En AT %M0.1, 500 ms
   "AlarmHorn_En" : Bool = PLC AlarmHorn_Out AT %M1.4, 500 ms
   "BrakeHand_PB" : Bool = PLC BrakeHand_PB AT %M28.2, 500 ms
   "BrakeOff_PB" : Bool = PLC BrakeOff_PB AT %M28.1, 500 ms
   "BrakeAuto_PB" : Bool = PLC BrakeAuto_PB AT %M28.3, 500 ms
   "StationIntHand_PB" : Bool = PLC StationIntHand_PB AT %M29.0, 500 ms
   "StationIntOff_PB" : Bool = PLC StationIntOff_PB AT %M28.7, 500 ms
   "StationIntAuto_PB" : Bool = PLC StationIntAuto_PB AT %M29.1, 500 ms
   "VFDHand_PB" : Bool = PLC VFDHand_PB AT %M93.5, 500 ms
   "VFDOff_PB" : Bool = PLC VFDOff_PB AT %M93.6, 500 ms
   "VFDAuto_PB" : Bool = PLC VFDAuto_PB AT %M102.1, 500 ms
   "BaffleHand_PB" : Bool = PLC BaffleHand_PB AT %M93.0, 500 ms
   "BaffleOff_PB" : Bool = PLC BaffleOff_PB AT %M93.1, 500 ms
   "BaffleAuto_PB" : Bool = PLC BaffleAuto_PB AT %M92.6, 500 ms
   "AlarmHornHand_PB" : Bool = PLC AlarmHornHand_PB AT %M28.5, 500 ms
   "AlarmHornOff_PB" : Bool = PLC AlarmHornOff_PB AT %M28.4, 500 ms
   "AlarmHornAuto_PB" : Bool = PLC AlarmHornAuto_PB AT %M28.6, 500 ms
   "ModeInt" : Int = PLC ModeInt AT %MW114, 500 ms
   "Brake_HOA" : Int = PLC Brake_HOA AT %MW32, 500 ms
   "StationInt_HOA" : Int = PLC StationInt_HOA AT %MW36, 500 ms
   "VFD_HOA" : Int = PLC VFD_HOA AT %MW100, 500 ms
   "Baffle_HOA" : Int = PLC Baffle_HOA AT %MW64, 500 ms
   "AlarmHorn_HOA" : Int = PLC AlarmHorn_HOA AT %MW34, 500 ms
   "HM_Minutes" : Int = PLC HM_Minutes AT %MW108, 500 ms
   "HM_Hours" : Int = PLC HM_Hours AT %MW110, 500 ms
   "HM_Days" : Int = PLC HM_Days AT %MW112, 500 ms
   "HMReset_PB" : Bool = PLC ResetHourmeter_PB AT %M103.1, 500 ms
   "FaultMode" : Bool = PLC FaultMode AT %M92.0, 500 ms
   "BrakeFailureDelay_SP" : Int = PLC BrakeFailureDelay_SP AT %MW60, 500 ms
   "Overcurrent_SP" : Int = PLC OvercurrentAlarm_SP AT %MW46, 500 ms
   "OvercurrentDelay_SP" : Int = PLC OvercurrentDelay_SP AT %MW44, 500 ms
   "RotorOverspeed_SP" : Int = PLC RotorOverspeedAlarm_SP AT %MW54, 500 ms
   "RotorOverspeedDelay_SP" : Int = PLC RotorOverspeedDelay_SP AT %MW52, 500 ms
   "HighOilTemp_SP" : Int = PLC HighOilTempAlarm_SP AT %MW50, 500 ms
   "HighOilTempDelay_SP" : Int = PLC HighOilTempDelay_SP AT %MW48, 500 ms
   "OilLowFlow_SP" : Int = PLC OilLowFlowAlarm_SP AT %MW42, 500 ms
   "OilLowFlowDelay_SP" : Int = PLC OilLowFlowDelay_SP AT %MW38, 500 ms
   "OilHighFlow_SP" : Int = PLC OilHighFlowAlarm_SP AT %MW58, 500 ms
   "OilHighFlowDelay_SP" : Int = PLC OilHighFlowDelay_SP AT %MW56, 500 ms
   "WarmupOilTemp_SP" : Int = PLC WarmupOilTemp_SP AT %MW74, 500 ms
   "WarmupDelay_SP" : Int = PLC WarmupOilTempDelay_SP AT %MW76, 500 ms
   "StabilizeCurrent_SP" : Int = PLC StabilizekW_SP AT %MW80, 500 ms
   "StabilizeDelay_SP" : Int = PLC StabilizeDelay_SP AT %MW82, 500 ms
   "CooldownOilTemp_SP" : Int = PLC CooldownOilTemp_SP AT %MW90, 500 ms
   "CooldownDelay_SP" : Int = PLC CooldownDelay_SP AT %MW86, 500 ms
   "VFDManual_SP" : Real = PLC VFDManual_SP AT %MD104, 500 ms
   "BaffleManual_SP" : Real = PLC BaffleManual_SP AT %MD96, 500 ms
   "ProgramLanguage" : Int = PLC ProgLang AT %MW12, 500 ms
   "LAD_PB" : Bool = PLC PB_LAD AT %M0.4, 500 ms
   "FBD_PB" : Bool = PLC PB_FBD AT %M0.6, 500 ms
   "SCL_PB" : Bool = PLC PB_SCL AT %M0.7, 500 ms
   "STL_PB" : Bool = PLC PB_STL AT %M1.0, 500 ms
   "Current" : Int = PLC Current AT %MW26, 500 ms
   "OilTemp" : Int = PLC OilTemp AT %MW20, 500 ms
   "OilFlow" : Int = PLC OilFlow AT %MW22, 500 ms
   "Baffle_Pct" : Int = PLC Baffle_Pct AT %MW16, 500 ms
   "VFD_Pct" : Int = PLC OilPumpVFDsp_Pct AT %MW14, 500 ms
   "RPM" : Int = PLC RPM AT %MW24, 500 ms
   "AlarmSilence" : Bool = PLC AlarmSilence AT %M40.0, 500 ms
   "AlarmReset" : Bool = PLC AlarmReset AT %M29.7, 500 ms
   "EStopNotify" : Bool = PLC EStopNotify AT %M41.7, 500 ms
   "BrakeFailureNotify" : Bool = PLC BrakeFailureNotify AT %M41.4, 500 ms
   "RotorOverspeedNotify" : Bool = PLC RotorOverspeedNotify AT %M41.0, 500 ms
   "OvercurrentNotify" : Bool = PLC OvercurrentNotify AT %M40.4, 500 ms
   "OilLowFlowNotify" : Bool = PLC OilLowFlowNotify AT %M40.2, 500 ms
   "OilHighFlowNotify" : Bool = PLC OilHighFlowNotify AT %M41.2, 500 ms
   "HighOilTempNotify" : Bool = PLC HighOilTempNotify AT %M40.6, 500 ms

discrete alarms
   1: 'E-Stop', class Errors, trigger "EStopNotify" bit 0
   2: 'Brake Failed', class Errors, trigger "BrakeFailureNotify" bit 0
   3: 'Overcurrent', class Errors, trigger "OvercurrentNotify" bit 0
   4: 'Rotor Overspeed', class Errors, trigger "RotorOverspeedNotify" bit 0
   5: 'High Oil Flow', class Errors, trigger "OilHighFlowNotify" bit 0
   6: 'Low Oil Flow', class Errors, trigger "OilLowFlowNotify" bit 0
   7: 'High Oil Temp', class Errors, trigger "HighOilTempNotify" bit 0

screen "Status" 500x500
   TextField "Text field_3" at 9,9 size 127x24; Text 'System Status'
   Button "Button_1" at 9,451 size 80x30; TextOff 'Main'
      on Click: ActivateScreen("Status", 0)
   Button "Button_2" at 117,451 size 80x30; TextOff 'Overview'
      on Click: ActivateScreen("Overview", 0)
   Button "Button_3" at 226,451 size 80x30; TextOff 'Alarms'
   Button "Button_4" at 334,451 size 80x30; TextOff 'Config'
   Group "Group_2" at 443,442 size 48x48
   TextField "Text field_4" at 255,48 size 229x38; Text 'Generation Mode'
      Visibility <- "ModeInt"
   TextField "Text field_5" at 349,48 size 134x38; Text 'Idle Mode'
      Visibility <- "ModeInt"
   TextField "Text field_6" at 287,48 size 196x38; Text 'Warmup Mode'
      Visibility <- "ModeInt"
   TextField "Text field_7" at 291,48 size 193x38; Text 'Stabilize Mode'
      Visibility <- "ModeInt"
   TextField "Text field_8" at 271,48 size 212x38; Text 'Cooldown Mode'
      Visibility <- "ModeInt"
   RoundButton "Round button_1" at 360,325 size 48x48; Text 'LAD'
      on PressLeft: SetBit("LAD_PB")
      on ReleaseLeft: ResetBit("LAD_PB")
   RoundButton "Round button_2" at 410,325 size 48x48; Text 'FBD'
      on PressLeft: SetBit("FBD_PB")
      on ReleaseLeft: ResetBit("FBD_PB")
   RoundButton "Round button_3" at 359,373 size 48x48; Text 'SCL'
      on PressLeft: SetBit("SCL_PB")
      on ReleaseLeft: ResetBit("SCL_PB")
   RoundButton "Round button_4" at 409,373 size 48x48; Text 'STL'
      on PressLeft: SetBit("STL_PB")
      on ReleaseLeft: ResetBit("STL_PB")
   RoundButton "Round button_5" at 33,325 size 98x98; Text 'START'
      on PressLeft: SetBit("SystemStart_PB")
      on ReleaseLeft: SetBit("SystemStart_PB")
   RoundButton "Round button_6" at 149,325 size 98x98; Text 'STOP'
      on PressLeft: SetBit("SystemStop_PB")
      on ReleaseLeft: SetBit("SystemStop_PB")
   IOField "I/O field_1" at 230,135 size 80x54; FormatPattern s99999
      ProcessValue <- "Current"
   TextField "Text field_13" at 105,149 size 73x24; Text 'Current:'
   TextField "Text field_14" at 326,149 size 28x24; Text 'kW'
   TextField "Text field_15" at 89,225 size 85x24; Text 'Interlock:'
   Group "Group_4" at 325,287 size 165x27
   Group "Group_3" at 222,225 size 93x30
   Button "Button_5" at 411,9 size 80x30; TextOff 'Exit App'
      on Click: StopRuntime(0)
   TextField "Text field_2" at 455,457 size 25x19; Text 'OK!'
   Group "Group_1" at 443,442 size 48x48
   Group "Group" at 443,442 size 48x48
      Visibility <- "FaultMode"
   TextField "Text field_1" at 444,457 size 47x19; Text 'Alarm!'
   TextField "Text field_9" at 344,288 size 145x26; Text 'Ladder Diagram'
      Visibility <- "ProgramLanguage"
   TextField "Text field_10" at 360,287 size 130x26; Text 'Function Block'
      Visibility <- "ProgramLanguage"
   TextField "Text field_11" at 325,288 size 164x26; Text 'Structured Control'
      Visibility <- "ProgramLanguage"
   TextField "Text field_12" at 357,288 size 132x26; Text 'Statement List'
      Visibility <- "ProgramLanguage"
   TextField "Text field_17" at 229,225 size 81x30; Text 'OFFLINE'
      Visibility <- "StationInt_En"
   TextField "Text field_16" at 222,225 size 93x30; Text 'ENGAGED'
      Visibility <- "StationInt_En"

screen "Overview" 500x500
   TextField "Text field_3" at 9,9 size 154x24; Text 'System Overview'
   Button "Button_1" at 9,451 size 80x30; TextOff 'Main'
      on Click: ActivateScreen("Status", 0)
   Button "Button_2" at 117,451 size 80x30; TextOff 'Overview'
      on Click: ActivateScreen("Overview", 0)
   Button "Button_3" at 226,451 size 80x30; TextOff 'Alarms'
   Button "Button_4" at 334,451 size 80x30; TextOff 'Config'
   Group "Group_2" at 443,442 size 48x48
   GraphicView "Graphic view_1" at 1,50 size 498x312; Picture "canvas"
   IOField "I/O field_1" at 11,336 size 80x45; FormatPattern 99999999
      ProcessValue <- "Baffle_Pct"
   TextField "Text field_4" at 23,384 size 60x19; Text 'Baffle %'
   IOField "I/O field_2" at 236,344 size 80x45; FormatPattern 99999999
      ProcessValue <- "RPM"
   TextField "Text field_5" at 260,390 size 31x19; Text 'RPM'
   IOField "I/O field_3" at 153,165 size 80x45; FormatPattern 99999999
      ProcessValue <- "VFD_Pct"
   TextField "Text field_6" at 151,210 size 87x19; Text 'Oil Pump %'
   Group "Group_7" at 265,66 size 135x32
   Group "Group_8" at 363,345 size 135x32
   Group "Group_9" at 17,49 size 48x48
      Visibility <- "EStopAlarm"
   Group "Group_10" at 76,49 size 48x48
      Visibility <- "BrakeFailureAlarm"
   Group "Group_11" at 135,49 size 48x48
      Visibility <- "RotorOverspeedAlarm"
   Group "Group_12" at 194,49 size 48x48
      Visibility <- "OvercurrentAlarm"
   Group "Group_13" at 108,102 size 48x48
      Visibility <- "OilLowFlowAlarm"
   Group "Group_14" at 167,102 size 48x48
      Visibility <- "OilHighFlowAlarm"
   Group "Group_15" at 49,102 size 48x48
      Visibility <- "HighOilTempAlarm"
   Group "Group_16" at 9,47 size 241x109
      Visibility <- "FaultMode"
   TextField "Text field_19" at 28,406 size 229x38; Text 'Generation Mode'
      Visibility <- "ModeInt"
   TextField "Text field_20" at 122,406 size 134x38; Text 'Idle Mode'
      Visibility <- "ModeInt"
   TextField "Text field_21" at 60,406 size 196x38; Text 'Warmup Mode'
      Visibility <- "ModeInt"
   TextField "Text field_22" at 64,406 size 193x38; Text 'Stabilize Mode'
      Visibility <- "ModeInt"
   TextField "Text field_23" at 44,406 size 212x38; Text 'Cooldown Mode'
      Visibility <- "ModeInt"
   Button "Button_5" at 411,9 size 80x30; TextOff 'Exit App'
      on Click: StopRuntime(0)
   IOField "I/O field_4" at 146,336 size 80x45; FormatPattern 99999999
      ProcessValue <- "OilTemp"
   TextField "Text field_24" at 155,383 size 66x19; Text 'Oil Temp'
   IOField "I/O field_5" at 345,383 size 80x45; FormatPattern 99999999
      ProcessValue <- "Current"
   TextField "Text field_25" at 339,428 size 92x19; Text 'Current (kW)'
   TextField "Text field_2" at 455,457 size 25x19; Text 'OK!'
   Group "Group_1" at 443,442 size 48x48
   Group "Group" at 443,442 size 48x48
      Visibility <- "FaultMode"
   TextField "Text field_1" at 444,457 size 47x19; Text 'Alarm!'
   TextField "Text field_8" at 378,352 size 106x19; Text 'Brake Released'
   TextField "Text field_7" at 376,352 size 109x19; Text 'Brake Engaged!'
   TextField "Text field_9" at 269,73 size 128x19; Text 'Interlock Engaged'
   TextField "Text field_10" at 287,73 size 91x19; Text 'No Interlock!'
   Group "Group_3" at 265,66 size 135x32
      Visibility <- "StationInt_En"
   Group "Group_4" at 265,66 size 135x32
      Visibility <- "StationInt_En"
   Group "Group_5" at 363,345 size 135x32
      Visibility <- "Brake_En"
   Group "Group_6" at 363,345 size 135x32
      Visibility <- "Brake_En"
   TextField "Text field_11" at 23,65 size 37x17; Text 'EStop'
   TextField "Text field_12" at 83,65 size 34x17; Text 'Brake'
   TextField "Text field_13" at 140,65 size 38x17; Text 'Speed'
   TextField "Text field_14" at 195,65 size 47x17; Text 'Current'
   TextField "Text field_15" at 115,118 size 34x17; Text 'LFlow'
   TextField "Text field_16" at 173,118 size 36x17; Text 'HFlow'
   TextField "Text field_17" at 51,118 size 44x17; Text 'HTemp'
   TextField "Text field_18" at 86,88 size 97x24; Text 'No Alarms.'

screen "Alarms" 500x500
   TextField "Text field_2" at 455,457 size 25x19; Text 'OK!'
   Group "Group_1" at 443,442 size 48x48
   Group "Group" at 443,442 size 48x48
      Visibility <- "FaultMode"
   TextField "Text field_1" at 444,457 size 47x19; Text 'Alarm!'
   TextField "Text field_3" at 9,9 size 174x24; Text 'Alarm Management'
   Button "Button_1" at 9,451 size 80x30; TextOff 'Main'
      on Click: ActivateScreen("Status", 0)
   Button "Button_2" at 117,451 size 80x30; TextOff 'Overview'
      on Click: ActivateScreen("Overview", 0)
   Button "Button_3" at 226,451 size 80x30; TextOff 'Alarms'
   Button "Button_4" at 334,451 size 80x30; TextOff 'Config'
   Group "Group_2" at 443,442 size 48x48
   AlarmControl "Alarm view_1" at 9,47 size 484x254
   RoundButton "Round button_1" at 285,347 size 74x74; Text 'SILENCE'
      on PressLeft: SetBit("AlarmSilence_PB")
      on ReleaseLeft: ResetBit("AlarmSilence_PB")
   RoundButton "Round button_2" at 393,347 size 74x74; Text 'RESET'
      on PressLeft: SetBit("AlarmReset_PB")
      on ReleaseLeft: ResetBit("AlarmReset_PB")
   TextField "Text field_4" at 317,309 size 116x22; Text 'Alarm Controls'
   Group "Group_3" at 17,320 size 48x48
      Visibility <- "EStopAlarm"
   Group "Group_4" at 76,320 size 48x48
      Visibility <- "BrakeFailureAlarm"
   Group "Group_5" at 135,320 size 48x48
      Visibility <- "RotorOverspeedAlarm"
   Group "Group_6" at 194,320 size 48x48
      Visibility <- "OvercurrentAlarm"
   Group "Group_8" at 108,373 size 48x48
      Visibility <- "OilLowFlowAlarm"
   Group "Group_9" at 167,373 size 48x48
      Visibility <- "OilHighFlowAlarm"
   Group "Group_7" at 49,373 size 48x48
      Visibility <- "HighOilTempAlarm"
   Group "Group_10" at 9,318 size 241x109
      Visibility <- "FaultMode"
   Button "Button_5" at 411,9 size 80x30; TextOff 'Exit App'
      on Click: StopRuntime(0)
   TextField "Text field_6" at 23,336 size 37x17; Text 'EStop'
   TextField "Text field_5" at 83,336 size 34x17; Text 'Brake'
   TextField "Text field_7" at 140,336 size 38x17; Text 'Speed'
   TextField "Text field_8" at 195,336 size 47x17; Text 'Current'
   TextField "Text field_9" at 51,389 size 44x17; Text 'HTemp'
   TextField "Text field_10" at 115,389 size 34x17; Text 'LFlow'
   TextField "Text field_11" at 173,389 size 36x17; Text 'HFlow'
   TextField "Text field_12" at 86,359 size 97x24; Text 'No Alarms.'

screen "Config" 500x500
   TextField "Text field_1" at 444,457 size 47x19; Text 'Alarm!'
   TextField "Text field_2" at 455,457 size 25x19; Text 'OK!'
   Group "Group_1" at 443,442 size 48x48
   Group "Group" at 443,442 size 48x48
      Visibility <- "FaultMode"
   Button "Button_1" at 9,451 size 80x30; TextOff 'Main'
      on Click: ActivateScreen("Status", 0)
   Button "Button_2" at 117,451 size 80x30; TextOff 'Overview'
      on Click: ActivateScreen("Overview", 0)
   Button "Button_3" at 226,451 size 80x30; TextOff 'Alarms'
   Button "Button_4" at 334,451 size 80x30; TextOff 'Config'
   Group "Group_2" at 443,442 size 48x48
   TextField "Text field_3" at 9,9 size 119x24; Text 'Configuration'
   IOField "I/O field_1" at 175,68 size 43x20; FormatPattern s99999
      ProcessValue <- "WarmupOilTemp_SP"
   TextField "Text field_4" at 80,46 size 89x17; Text 'Process Values'
   TextField "Text field_5" at 76,70 size 93x17; Text 'Warmup Temp'
   TextField "Text field_6" at 78,95 size 92x17; Text 'Warmup Delay'
   TextField "Text field_7" at 92,118 size 78x17; Text 'Current (kw)'
   TextField "Text field_8" at 84,143 size 85x17; Text 'Stabilize Delay'
   TextField "Text field_9" at 70,168 size 100x17; Text 'Cooldown Temp'
   TextField "Text field_10" at 70,196 size 99x17; Text 'Cooldown Delay'
   IOField "I/O field_2" at 175,93 size 43x20; FormatPattern s99999
      ProcessValue <- "WarmupDelay_SP"
   IOField "I/O field_3" at 175,118 size 43x20; FormatPattern s99999
      ProcessValue <- "StabilizeCurrent_SP"
   IOField "I/O field_4" at 175,143 size 43x20; FormatPattern s99999
      ProcessValue <- "StabilizeDelay_SP"
   IOField "I/O field_5" at 175,168 size 43x20; FormatPattern s99999
      ProcessValue <- "CooldownOilTemp_SP"
   IOField "I/O field_6" at 175,195 size 43x20; FormatPattern s99999
      ProcessValue <- "CooldownDelay_SP"
   IOField "I/O field_7" at 431,69 size 43x20; FormatPattern s99999
      ProcessValue <- "BrakeFailureDelay_SP"
   TextField "Text field_11" at 351,49 size 76x17; Text 'Alarm Values'
   TextField "Text field_12" at 313,69 size 114x17; Text 'Brake Failure Delay'
   TextField "Text field_13" at 291,94 size 136x17; Text 'Rotor Overspeed RPM'
   TextField "Text field_14" at 284,119 size 143x17; Text 'Rotor Overspeed Delay'
   TextField "Text field_15" at 306,143 size 120x17; Text 'High Temp Degrees'
   TextField "Text field_16" at 322,171 size 104x17; Text 'High Temp Delay'
   IOField "I/O field_8" at 431,94 size 43x20; FormatPattern s99999
      ProcessValue <- "RotorOverspeed_SP"
   IOField "I/O field_9" at 431,119 size 43x20; FormatPattern s99999
      ProcessValue <- "RotorOverspeedDelay_SP"
   IOField "I/O field_10" at 431,144 size 43x20; FormatPattern s99999
      ProcessValue <- "HighOilTemp_SP"
   IOField "I/O field_11" at 431,171 size 43x20; FormatPattern s99999
      ProcessValue <- "HighOilTempDelay_SP"
   TextField "Text field_17" at 339,197 size 87x17; Text 'Low Flow GPM'
   TextField "Text field_18" at 332,223 size 94x17; Text 'Low Flow Delay'
   TextField "Text field_19" at 336,253 size 89x17; Text 'High Flow GPM'
   TextField "Text field_20" at 330,281 size 96x17; Text 'High Flow Delay'
   IOField "I/O field_12" at 431,197 size 43x20; FormatPattern s99999
      ProcessValue <- "OilLowFlow_SP"
   IOField "I/O field_13" at 431,223 size 43x20; FormatPattern s99999
      ProcessValue <- "OilLowFlowDelay_SP"
   IOField "I/O field_14" at 431,253 size 43x20; FormatPattern s99999
      ProcessValue <- "OilHighFlow_SP"
   IOField "I/O field_15" at 431,282 size 43x20; FormatPattern s99999
      ProcessValue <- "OilHighFlowDelay_SP"
   TextField "Text field_21" at 324,313 size 100x17; Text 'Overcurrent kW'
   TextField "Text field_22" at 312,342 size 113x17; Text 'Overcurrent Delay'
   IOField "I/O field_16" at 431,313 size 43x20; FormatPattern s99999
      ProcessValue <- "Overcurrent_SP"
   IOField "I/O field_17" at 431,342 size 43x20; FormatPattern s99999
      ProcessValue <- "OvercurrentDelay_SP"
   TextField "Text field_23" at 89,283 size 82x17; Text 'HOA Controls'
   TextField "Text field_24" at 53,307 size 68x17; Text 'Alarm Horn'
   TextField "Text field_25" at 87,337 size 34x17; Text 'Brake'
   TextField "Text field_26" at 22,364 size 100x17; Text 'Station Interlock'
   TextField "Text field_27" at 90,391 size 32x17; Text 'Baffle'
   TextField "Text field_28" at 39,415 size 83x17; Text 'Oil Pump VFD'
   Button "Button_5" at 127,306 size 20x20; TextOff 'H'
      on PressLeft: SetBit("AlarmHornHand_PB")
      on ReleaseLeft: SetBit("AlarmHornHand_PB")
   Button "Button_6" at 156,306 size 20x20; TextOff 'O'
      on PressLeft: SetBit("AlarmHornOff_PB")
      on ReleaseLeft: SetBit("AlarmHornOff_PB")
   Button "Button_7" at 185,306 size 20x20; TextOff 'A'
      on PressLeft: SetBit("AlarmHornAuto_PB")
      on ReleaseLeft: SetBit("AlarmHornAuto_PB")
   Button "Button_8" at 127,334 size 20x20; TextOff 'H'
      on PressLeft: SetBit("BrakeHand_PB")
      on ReleaseLeft: SetBit("BrakeHand_PB")
   Button "Button_9" at 156,334 size 20x20; TextOff 'O'
      on PressLeft: SetBit("BrakeOff_PB")
      on ReleaseLeft: SetBit("BrakeOff_PB")
   Button "Button_10" at 185,334 size 20x20; TextOff 'A'
      on PressLeft: SetBit("BrakeAuto_PB")
      on ReleaseLeft: SetBit("BrakeAuto_PB")
   Button "Button_11" at 127,362 size 20x20; TextOff 'H'
      on PressLeft: SetBit("StationIntHand_PB")
      on ReleaseLeft: SetBit("StationIntHand_PB")
   Button "Button_12" at 156,362 size 20x20; TextOff 'O'
      on PressLeft: SetBit("StationIntOff_PB")
      on ReleaseLeft: SetBit("StationIntOff_PB")
   Button "Button_13" at 185,362 size 20x20; TextOff 'A'
      on PressLeft: SetBit("StationIntAuto_PB")
      on ReleaseLeft: SetBit("StationIntAuto_PB")
   Rectangle "Rectangle_4" at 224,306 size 20x20
      Visibility <- "AlarmHorn_HOA"
   Button "Button_14" at 127,389 size 20x20; TextOff 'H'
      on PressLeft: SetBit("BaffleHand_PB")
      on ReleaseLeft: SetBit("BaffleHand_PB")
   Button "Button_15" at 156,389 size 20x20; TextOff 'O'
      on PressLeft: SetBit("BaffleOff_PB")
      on ReleaseLeft: SetBit("BaffleOff_PB")
   Button "Button_16" at 185,389 size 20x20; TextOff 'A'
      on PressLeft: SetBit("BaffleAuto_PB")
      on ReleaseLeft: SetBit("BaffleAuto_PB")
   Button "Button_17" at 127,415 size 20x20; TextOff 'H'
      on PressLeft: SetBit("VFDHand_PB")
      on ReleaseLeft: SetBit("VFDHand_PB")
   Button "Button_18" at 156,415 size 20x20; TextOff 'O'
      on PressLeft: SetBit("VFDOff_PB")
      on ReleaseLeft: SetBit("VFDOff_PB")
   Button "Button_19" at 185,415 size 20x20; TextOff 'A'
      on PressLeft: SetBit("VFDAuto_PB")
      on ReleaseLeft: SetBit("VFDAuto_PB")
   Rectangle "Rectangle_5" at 224,334 size 20x20
      Visibility <- "Brake_HOA"
   Rectangle "Rectangle_6" at 224,362 size 20x20
      Visibility <- "StationInt_HOA"
   Rectangle "Rectangle_7" at 224,389 size 20x20
      Visibility <- "Baffle_HOA"
   Rectangle "Rectangle_8" at 224,415 size 20x20
      Visibility <- "VFD_HOA"
   Rectangle "Rectangle_9" at 224,306 size 20x20
      Visibility <- "AlarmHorn_HOA"
   Rectangle "Rectangle_10" at 224,306 size 20x20
      Visibility <- "AlarmHorn_HOA"
   Rectangle "Rectangle_11" at 224,334 size 20x20
      Visibility <- "Brake_HOA"
   Rectangle "Rectangle_12" at 224,334 size 20x20
      Visibility <- "Brake_HOA"
   Rectangle "Rectangle_13" at 224,362 size 20x20
      Visibility <- "StationInt_HOA"
   Rectangle "Rectangle_14" at 224,389 size 20x20
      Visibility <- "Baffle_HOA"
   Rectangle "Rectangle_15" at 224,415 size 20x20
      Visibility <- "VFD_HOA"
   Rectangle "Rectangle_16" at 224,362 size 20x20
      Visibility <- "StationInt_HOA"
   Rectangle "Rectangle_17" at 224,389 size 20x20
      Visibility <- "Baffle_HOA"
   Rectangle "Rectangle_18" at 224,415 size 20x20
      Visibility <- "VFD_HOA"
   TextField "Text field_29" at 72,221 size 98x17; Text 'Baffle Manual SP'
   TextField "Text field_30" at 19,249 size 149x17; Text 'Oil Pump VFD Manual SP'
   IOField "I/O field_18" at 175,221 size 43x20; FormatPattern s999999999.999
      ProcessValue <- "BaffleManual_SP"
   IOField "I/O field_19" at 175,248 size 43x20; FormatPattern s999999999.999
      ProcessValue <- "VFDManual_SP"
   TextField "Text field_31" at 339,381 size 66x17; Text 'Hourmeter'
   Button "Button_20" at 455,406 size 20x20; TextOff 'R'
      on PressLeft: SetBit("HMReset_PB")
      on ReleaseLeft: SetBit("HMReset_PB")
   IOField "I/O field_20" at 282,406 size 43x20; FormatPattern s99999
      ProcessValue <- "HM_Days"
   TextField "Text field_32" at 270,406 size 10x17; Text 'D'
   IOField "I/O field_21" at 345,406 size 43x20; FormatPattern s99999
      ProcessValue <- "HM_Hours"
   TextField "Text field_33" at 333,406 size 10x17; Text 'H'
   IOField "I/O field_22" at 408,406 size 43x20; FormatPattern s99999
      ProcessValue <- "HM_Minutes"
   TextField "Text field_34" at 396,406 size 10x17; Text 'M'
   Button "Button_21" at 411,9 size 80x30; TextOff 'Exit App'
      on Click: StopRuntime(0)
*)